FUNCTION_BLOCK FB_ADD
VAR_INPUT
	in1,in2:INT;
END_VAR
VAR_OUTPUT
	out:INT;
END_VAR
VAR
END_VAR

out:=in1+in2;

END_FUNCTION_BLOCK

(* stored: Version 1.1.0.1, ProductVersion 3.1.4024.11
   POU FB_ADD: Id {720b20e9-9fd8-44ca-8bf9-6b397915c24d}, SpecialFunc None *)
